// TIA Portal V17 export
// export: Created 2025-03-07T09:19:08.2781851Z, ExportSetting WithDefaults, DisplayName Totally Integrated Automation Portal, DisplayVersion V17 Update 8, DisplayName TIA Portal Openness, DisplayVersion V17 Update 8, DisplayName TIA Portal Version Control Interface, DisplayVersion V17, DisplayName SINAMICS Startdrive Advanced, DisplayVersion V17 SP2, DisplayName SINAMICS Startdrive G110M, G120, G120C, G120D, G120P, G115D, DisplayVersion V17 SP2, DisplayName SINAMICS Startdrive G130, G150, S120, S150, SINAMICS MV, S210, DisplayVersion V17 SP2, DisplayName STEP 7 Professional, DisplayVersion V17 Update 8, DisplayName SINUMERIK ONE STEP 7 Toolbox, DisplayVersion V17 Update 12, DisplayName SINUMERIK 840D sl STEP 7 Toolbox, DisplayVersion V17 Update 12, DisplayName STEP 7 Safety, DisplayVersion V17 Update 6, DisplayName WinCC Advanced, DisplayVersion V17 Update 8
FUNCTION "FC10300_PT100_SENSOR_VALUES" : Void   // FC10300, LAD
{ S7_Optimized_Access := 'TRUE' }
VERSION : 0.1
// stored: AutoNumber false, IsIECCheckEnabled false, SetENOAutomatically false, UDAEnableTagReadback false
BEGIN

REGION Network 1: UNIT 01 PT100 SENSORS
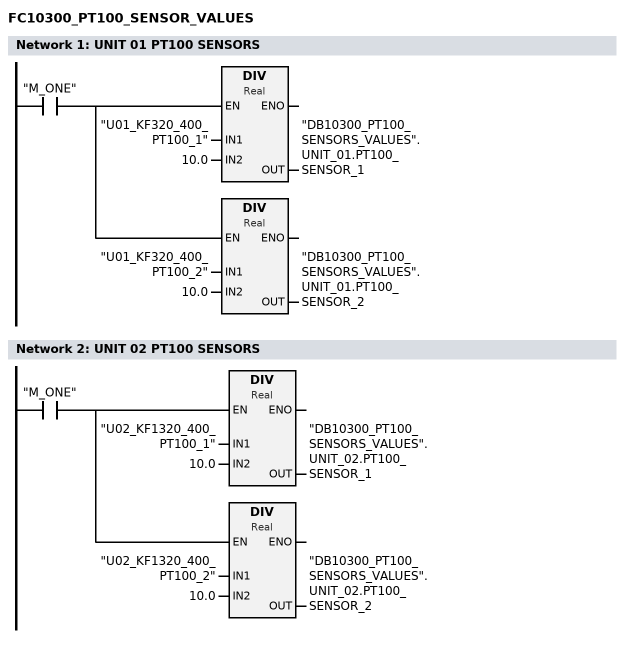
   RUNG wire#powerrail
      Contact( "M_ONE" )
      wire#w1
      { S7_Templates := "SrcType := Real" } Div(in1 := "U01_KF320_400_PT100_1", in2 := 10.0, out => "DB10300_PT100_SENSORS_VALUES".UNIT_01.PT100_SENSOR_1)
   END_RUNG
   RUNG wire#w1
      { S7_Templates := "SrcType := Real" } Div(in1 := "U01_KF320_400_PT100_2", in2 := 10.0, out => "DB10300_PT100_SENSORS_VALUES".UNIT_01.PT100_SENSOR_2)
   END_RUNG
   // the same network as SCL:
   IF "M_ONE" THEN
       "DB10300_PT100_SENSORS_VALUES".UNIT_01.PT100_SENSOR_1 := "U01_KF320_400_PT100_1" / 10.0;
       "DB10300_PT100_SENSORS_VALUES".UNIT_01.PT100_SENSOR_2 := "U01_KF320_400_PT100_2" / 10.0;
   END_IF;
END_REGION

REGION Network 2: UNIT 02 PT100 SENSORS
   RUNG wire#powerrail
      Contact( "M_ONE" )
      wire#w1
      { S7_Templates := "SrcType := Real" } Div(in1 := "U02_KF1320_400_PT100_1", in2 := 10.0, out => "DB10300_PT100_SENSORS_VALUES".UNIT_02.PT100_SENSOR_1)
   END_RUNG
   RUNG wire#w1
      { S7_Templates := "SrcType := Real" } Div(in1 := "U02_KF1320_400_PT100_2", in2 := 10.0, out => "DB10300_PT100_SENSORS_VALUES".UNIT_02.PT100_SENSOR_2)
   END_RUNG
   // the same network as SCL:
   IF "M_ONE" THEN
       "DB10300_PT100_SENSORS_VALUES".UNIT_02.PT100_SENSOR_1 := "U02_KF1320_400_PT100_1" / 10.0;
       "DB10300_PT100_SENSORS_VALUES".UNIT_02.PT100_SENSOR_2 := "U02_KF1320_400_PT100_2" / 10.0;
   END_IF;
END_REGION
END_FUNCTION
